{attribute 'qualified_only'}
{attribute 'strict'}
TYPE MovementDirection :
(
	TowardsSensor := 1,
	AwayFromSensor := 0
);
END_TYPE

(* stored: Version 1.1.0.1, ProductVersion 3.1.4024.13
   EnumerationTextList MovementDirection: Id {f3837e44-c460-4148-a488-3f505e0bf404} *)
